VAR_GLOBAL
	bGlobalReset		: BOOL;
	bButtonManStart 	: BOOL;
	bButtonAutoStart	: BOOL;
	nInputMachineIdx	: UINT;
	nInputStationIdx	: UINT;
	nInputLeakTestIdx	: UINT;
	
	bButtonReset		: BOOL;
	bButtonSaveRecipes	: BOOL;
	bButtonLoadLastSavedRecipes	: BOOL;
END_VAR

(* stored: Version 1.1.0.1
   GVL GVL_TcHmiControl: Id {cd6eb97a-f3b5-020e-2085-6ba74ac78815} *)
